FUNCTION_BLOCK FB_TempSensPt100 IMPLEMENTS I_TempSens
VAR_INPUT
END_VAR
VAR_OUTPUT
END_VAR
VAR
	Temp	:	REAL;
	TempRaw	AT %I*	:	INT;
	ConvFac : INT := 10;	//Conversion factor
END_VAR

METHOD Run : BOOL
Temp := INT_TO_REAL(TempRaw)/ConvFac;
END_METHOD

PROPERTY Temperature : REAL
GET
Temperature := Temp;
END_GET
SET
Temp := Temperature;
END_SET
END_PROPERTY

END_FUNCTION_BLOCK

(* stored: Version 1.1.0.1, ProductVersion 3.1.4022.10
   POU FB_TempSensPt100: Id {60e11487-1969-4eb3-8d78-2657500a42bc}, SpecialFunc None
   Method Run: Id {5e069eca-69e5-4426-bff7-45108ac3798c}
   Property Temperature: Id {7d5851d0-8b9c-424c-8d6b-fb269c5d74eb}
   Get Get: Id {574153b9-daa8-4f80-9414-e97e59bda2b9}
   Set Set: Id {e435d3b7-c16b-4b91-8e3e-60643b2418da} *)
